(* IEC 61131-3 sources: Word/plc-course/11-program-organization/labs/solutions, 3 files *)

(* ---- 11-1-motor-fb.st ---- *)
(* Lab 11-1: A reusable motor function block, used three times.
   Module 11 (Program organisation). REFERENCE SOLUTION - try the lab yourself first.

   A chemical dosing room has two dosing pumps and an extract fan. One
   function block type, FB_Motor, is written and tested once, then used for
   all three motors. Each instance (Pump1, Pump2, Fan1) has its own memory:
   its own seal-in, its own feedback timer and its own fault latch. *)

FUNCTION_BLOCK FB_Motor
  (* ------------------------------------------------------------------
     FB_Motor - direct-on-line motor with run feedback supervision.

     Behaviour
       - Start (TRUE) switches RunCmd on; RunCmd then holds itself on.
       - Stop, loss of InterlockOK, or a Fault switch RunCmd off. Stop wins
         over Start. The motor never restarts on its own: after a stop, an
         interlock trip or a reset it needs a new Start.
       - RunFb must agree with RunCmd. If they disagree for longer than
         FbTimeout (failed to start, lost feedback while running, or running
         without a command) Fault latches and RunCmd switches off.
       - Reset clears Fault. It does not restart the motor. If the cause is
         still there, the fault comes straight back.
       - Running = commanded AND feedback present ("proven running").
       - RunSeconds counts seconds of proven running (maintenance hours).
         It uses a 1 s timer that restarts every second, so it runs about
         one scan per second slow (1 % at a 10 ms scan). Good enough for
         maintenance hours, not for billing.

     The FB contains no I/O addresses. The calling program maps its inputs
     and outputs to real signals, so the same FB serves any motor.

     Version history
       1.0  first release (Lab 11-1)
     ------------------------------------------------------------------ *)
  VAR_INPUT
    Start       : BOOL;          (* start request, TRUE = start (pulse or held) *)
    Stop        : BOOL;          (* stop request, TRUE = stop; wins over Start *)
    InterlockOK : BOOL;          (* TRUE = allowed to run. No default TRUE on purpose:
                                    a forgotten connection must stop the motor,
                                    not bypass the interlock *)
    RunFb       : BOOL;          (* run feedback: contactor auxiliary contact,
                                    flow switch or airflow switch *)
    Reset       : BOOL;          (* fault reset *)
    FbTimeout   : TIME := T#2s;  (* how long RunFb may disagree with RunCmd *)
  END_VAR
  VAR_OUTPUT
    RunCmd      : BOOL;          (* command to the contactor coil *)
    Running     : BOOL;          (* proven running: RunCmd AND RunFb *)
    Fault       : BOOL;          (* latched feedback fault; needs Reset *)
    RunSeconds  : DINT;          (* extension: seconds of proven running *)
  END_VAR
  VAR
    FbCheck     : TON;           (* feedback discrepancy timer (a multi-instance) *)
    SecondTick  : TON;           (* 1 s time base for RunSeconds *)
  END_VAR

  (* 1. Reset. Checked first, so the discrepancy check further down can set
        the fault again in the same scan if its cause is still present. *)
  IF Reset THEN
    Fault := FALSE;
  END_IF;

  (* 2. Run command: seal-in with stop priority. Stop, interlock and fault
        are tested first, so none of them can be overridden by Start. *)
  IF Stop OR NOT InterlockOK OR Fault THEN
    RunCmd := FALSE;
  ELSIF Start THEN
    RunCmd := TRUE;
  END_IF;

  (* 3. Feedback supervision. XOR is TRUE whenever command and feedback
        disagree: failed to start, feedback lost while running, or running
        without a command (welded contactor, motor run in "hand"). The timer
        restarts every time they agree again. *)
  FbCheck(IN := RunCmd XOR RunFb, PT := FbTimeout);
  IF FbCheck.Q THEN
    Fault := TRUE;
    RunCmd := FALSE;
  END_IF;

  (* 4. Status *)
  Running := RunCmd AND RunFb;

  (* 5. Run-time accumulation (extension). The timer is restarted in the
        same scan that it finishes, so only one scan per second is lost. *)
  SecondTick(IN := Running, PT := T#1s);
  IF SecondTick.Q THEN
    RunSeconds := RunSeconds + 1;
    SecondTick(IN := FALSE);
  END_IF;
END_FUNCTION_BLOCK

PROGRAM DosingRoom
  VAR (* inputs *)
    Pump1StartPB   AT %IX0.0 : BOOL;  (* Pump 1 start push-button, NO *)
    Pump1StopPB_NC AT %IX0.1 : BOOL;  (* Pump 1 stop push-button, NC: TRUE while not pressed *)
    Pump1RunFb     AT %IX0.2 : BOOL;  (* Pump 1 contactor auxiliary contact: TRUE = contactor in *)
    Pump2StartPB   AT %IX0.3 : BOOL;  (* Pump 2 start push-button, NO *)
    Pump2StopPB_NC AT %IX0.4 : BOOL;  (* Pump 2 stop push-button, NC *)
    Pump2RunFb     AT %IX0.5 : BOOL;  (* Pump 2 contactor auxiliary contact *)
    Fan1StartPB    AT %IX0.6 : BOOL;  (* Extract fan start push-button, NO *)
    Fan1StopPB_NC  AT %IX0.7 : BOOL;  (* Extract fan stop push-button, NC *)
    Fan1AirflowSw  AT %IX1.0 : BOOL;  (* Extract duct airflow switch: TRUE = air moving *)
    TankLowLow_NC  AT %IX1.1 : BOOL;  (* Day-tank low-low level switch, fail-safe:
                                         TRUE = level healthy, FALSE = low-low or wire break *)
    ResetPB        AT %IX1.2 : BOOL;  (* Fault reset push-button, NO *)
  END_VAR
  VAR (* outputs *)
    Pump1Contactor AT %QX0.0 : BOOL;  (* Pump 1 contactor coil *)
    Pump2Contactor AT %QX0.1 : BOOL;  (* Pump 2 contactor coil *)
    Fan1Contactor  AT %QX0.2 : BOOL;  (* Extract fan contactor coil *)
    FaultLamp      AT %QX0.3 : BOOL;  (* Common "motor fault" lamp *)
  END_VAR
  VAR (* one instance of FB_Motor per motor *)
    Pump1 : FB_Motor;
    Pump2 : FB_Motor;
    Fan1  : FB_Motor;
  END_VAR

  (* The fan is called first because the pumps use its Running status.
     Calling it after the pumps would also work, one scan later. *)
  Fan1(Start       := Fan1StartPB,
       Stop        := NOT Fan1StopPB_NC,   (* polarity is handled here, not in the FB *)
       InterlockOK := TRUE,                (* the fan has no process interlock *)
       RunFb       := Fan1AirflowSw,
       Reset       := ResetPB,
       FbTimeout   := T#5s);               (* an airflow switch needs a few seconds to prove *)
  Fan1Contactor := Fan1.RunCmd;

  (* Dosing pumps may run only while the extract fan is PROVEN running and
     the day tank is above low-low. Fan1.Running, not Fan1.RunCmd: a fan
     that has been told to run but moves no air does not ventilate the room. *)
  Pump1(Start       := Pump1StartPB,
        Stop        := NOT Pump1StopPB_NC,
        InterlockOK := Fan1.Running AND TankLowLow_NC,
        RunFb       := Pump1RunFb,
        Reset       := ResetPB);           (* FbTimeout left at its 2 s default *)
  Pump1Contactor := Pump1.RunCmd;

  Pump2(Start       := Pump2StartPB,
        Stop        := NOT Pump2StopPB_NC,
        InterlockOK := Fan1.Running AND TankLowLow_NC,
        RunFb       := Pump2RunFb,
        Reset       := ResetPB);
  Pump2Contactor := Pump2.RunCmd;

  FaultLamp := Pump1.Fault OR Pump2.Fault OR Fan1.Fault;
END_PROGRAM

CONFIGURATION Config0
  RESOURCE Res0 ON PLC
    TASK MainTask(INTERVAL := T#10ms, PRIORITY := 0);
    PROGRAM Inst0 WITH MainTask : DosingRoom;
  END_RESOURCE
END_CONFIGURATION

(* ---- 11-2-valve-fb.st ---- *)
(* Lab 11-2: A reusable on/off valve function block with limit switches.
   Module 11 (Program organisation). REFERENCE SOLUTION - try the lab yourself first.

   Two spring-return pneumatic valves on a reactor use the same FB_Valve:
     XV101  reactor feed valve      fail CLOSED (loss of air/power stops the feed)
     XV102  jacket cooling valve    fail OPEN   (loss of air/power keeps cooling on)
   The FB is told which way its valve fails and works out the solenoid state
   for itself. Training exercise only: a real reactor trip belongs in a
   safety instrumented system, not in basic control logic (Module 20). *)

FUNCTION_BLOCK FB_Valve
  (* ------------------------------------------------------------------
     FB_Valve - single-solenoid, spring-return on/off valve with open and
     closed limit switches (ZSO / ZSC).

     Behaviour
       - OpenCmd TRUE = open the valve, FALSE = close it (a level command,
         as a sequence or HMI would give it).
       - FailOpen says where the spring takes the valve when the solenoid is
         de-energised. The solenoid is energised to move the valve AWAY from
         that fail position:  Solenoid = OpenCmd XOR FailOpen.
       - IsOpen / IsClosed are only TRUE when exactly one limit switch is made.
       - TravelFault latches if the valve is not in the commanded end position
         for longer than TravelTime. The timer restarts whenever the command
         changes, so a reversal mid-stroke gets a full TravelTime. It also
         catches a valve that drifts out of position with no command change
         (for example loss of instrument air).
       - LimitFault latches if both limit switches are made together for
         500 ms (a switch, adjustment or wiring fault; the filter ignores a
         momentary overlap).
       - On any fault the solenoid is de-energised, so the valve goes to its
         fail position, and stays there until Reset.
       - Reset clears both faults. After a reset the valve follows OpenCmd
         again and gets a fresh TravelTime. If a fault's cause is still
         present the fault comes back.

     Version history
       1.0  first release (Lab 11-2)
     ------------------------------------------------------------------ *)
  VAR_INPUT
    OpenCmd    : BOOL;            (* TRUE = open, FALSE = close *)
    OpenLS     : BOOL;            (* open limit switch (ZSO), TRUE = fully open *)
    ClosedLS   : BOOL;            (* closed limit switch (ZSC), TRUE = fully closed *)
    Reset      : BOOL;            (* fault reset *)
    FailOpen   : BOOL;            (* configuration: TRUE = spring opens the valve *)
    TravelTime : TIME := T#10s;   (* longest acceptable stroke *)
  END_VAR
  VAR_OUTPUT
    Solenoid    : BOOL;           (* solenoid output *)
    IsOpen      : BOOL;           (* confirmed open *)
    IsClosed    : BOOL;           (* confirmed closed *)
    TravelFault : BOOL;           (* latched: did not reach / stay in position *)
    LimitFault  : BOOL;           (* latched: both limit switches made *)
    Fault       : BOOL;           (* TravelFault OR LimitFault *)
  END_VAR
  VAR
    TravelTmr  : TON;
    LimitTmr   : TON;
    InPosition : BOOL;            (* at the end position the command asks for *)
    LastCmd    : BOOL;            (* OpenCmd on the previous call *)
  END_VAR

  (* 1. Decode the limit switches. Exactly one must be made. *)
  IsOpen := OpenLS AND NOT ClosedLS;
  IsClosed := ClosedLS AND NOT OpenLS;

  (* 2. Reset first, so a fault whose cause is still present re-latches below. *)
  IF Reset THEN
    TravelFault := FALSE;
    LimitFault := FALSE;
  END_IF;

  (* 3. Limit switch discrepancy: both made is physically impossible. *)
  LimitTmr(IN := OpenLS AND ClosedLS, PT := T#500ms);
  IF LimitTmr.Q THEN
    LimitFault := TRUE;
  END_IF;

  (* 4. Travel supervision. The timer runs while the valve is not where it
        was told to be. It is held off for one call when the command changes
        (so it restarts) and while a fault is latched (so that a reset gives
        the valve a fresh TravelTime instead of an instant re-trip). *)
  IF OpenCmd THEN
    InPosition := IsOpen;
  ELSE
    InPosition := IsClosed;
  END_IF;
  TravelTmr(IN := NOT InPosition AND (OpenCmd = LastCmd)
                  AND NOT TravelFault AND NOT LimitFault,
            PT := TravelTime);
  IF TravelTmr.Q THEN
    TravelFault := TRUE;
  END_IF;
  LastCmd := OpenCmd;

  (* 5. Outputs. On a fault the solenoid drops out: the spring takes the
        valve to its fail (safe) position, whichever way that is. *)
  Fault := TravelFault OR LimitFault;
  IF Fault THEN
    Solenoid := FALSE;
  ELSE
    Solenoid := OpenCmd XOR FailOpen;
  END_IF;
END_FUNCTION_BLOCK

PROGRAM ReactorValves
  VAR (* inputs *)
    XV101_OpenSw AT %IX0.0 : BOOL;  (* XV-101 panel selector: TRUE = OPEN, FALSE = CLOSE *)
    XV101_ZSO    AT %IX0.1 : BOOL;  (* XV-101 open limit switch *)
    XV101_ZSC    AT %IX0.2 : BOOL;  (* XV-101 closed limit switch *)
    XV102_OpenSw AT %IX0.3 : BOOL;  (* XV-102 panel selector: TRUE = OPEN, FALSE = CLOSE *)
    XV102_ZSO    AT %IX0.4 : BOOL;  (* XV-102 open limit switch *)
    XV102_ZSC    AT %IX0.5 : BOOL;  (* XV-102 closed limit switch *)
    ResetPB      AT %IX0.6 : BOOL;  (* Fault reset push-button, NO *)
  END_VAR
  VAR (* outputs *)
    XV101_SOL    AT %QX0.0 : BOOL;  (* XV-101 solenoid: energise to OPEN (fail closed) *)
    XV102_SOL    AT %QX0.1 : BOOL;  (* XV-102 solenoid: energise to CLOSE (fail open) *)
    FaultLamp    AT %QX0.2 : BOOL;  (* Common "valve fault" lamp *)
  END_VAR
  VAR (* device instances *)
    XV101 : FB_Valve;               (* reactor feed valve *)
    XV102 : FB_Valve;               (* jacket cooling-water valve *)
  END_VAR

  XV101(OpenCmd    := XV101_OpenSw,
        OpenLS     := XV101_ZSO,
        ClosedLS   := XV101_ZSC,
        Reset      := ResetPB,
        FailOpen   := FALSE,        (* spring closes it: stop feeding on loss of air *)
        TravelTime := T#5s);
  XV101_SOL := XV101.Solenoid;

  XV102(OpenCmd    := XV102_OpenSw,
        OpenLS     := XV102_ZSO,
        ClosedLS   := XV102_ZSC,
        Reset      := ResetPB,
        FailOpen   := TRUE,         (* spring opens it: keep cooling on loss of air *)
        TravelTime := T#8s);        (* larger valve, slower actuator *)
  XV102_SOL := XV102.Solenoid;

  FaultLamp := XV101.Fault OR XV102.Fault;
END_PROGRAM

CONFIGURATION Config0
  RESOURCE Res0 ON PLC
    TASK MainTask(INTERVAL := T#10ms, PRIORITY := 0);
    PROGRAM Inst0 WITH MainTask : ReactorValves;
  END_RESOURCE
END_CONFIGURATION

(* ---- 11-3-function-library.st ---- *)
(* Lab 11-3: A small function library and a statistics FB using VAR_IN_OUT.
   Module 11 (Program organisation). REFERENCE SOLUTION - try the lab yourself first.

   A filling line has two filling heads, each with its own check-weigher.
   One instance of FB_SampleStats per head judges each weight against the
   limits and adds it to ONE shared statistics record, LineStats, which the
   instances reach through VAR_IN_OUT. Two FUNCTIONs form a small reusable
   library: F_InRange (limit check) and F_Deadband (report-by-exception). *)

TYPE
  ST_Stats :
  STRUCT
    Count    : DINT;    (* samples since the last clear *)
    InSpec   : DINT;    (* samples inside the limits *)
    OutSpec  : DINT;    (* samples outside the limits *)
    MinValue : REAL;    (* smallest sample since the last clear *)
    MaxValue : REAL;    (* largest sample since the last clear *)
    Sum      : LREAL;   (* running total. LREAL: a REAL has only about 7 significant
                           digits. Once a REAL total passes about 8.4 million (some
                           17,000 samples of 500 g) it can only change in whole grams,
                           so every new weight would be rounded to a whole gram *)
    Mean     : REAL;    (* Sum / Count *)
  END_STRUCT;
END_TYPE

FUNCTION F_InRange : BOOL
  (* TRUE when Low <= Value <= High (both limits included).
     If Low > High the range is empty and the result is always FALSE, so a
     limit entry mistake shows up as "everything out of range" rather than
     being silently repaired. No memory: same inputs, same answer. *)
  VAR_INPUT
    Value : REAL;
    Low   : REAL;
    High  : REAL;
  END_VAR
  F_InRange := (Value >= Low) AND (Value <= High);
END_FUNCTION

FUNCTION F_Deadband : REAL
  (* Report-by-exception: returns NewValue when it differs from OldValue by
     Band or more, otherwise returns OldValue unchanged.
     A function has no memory, so the CALLER keeps the last reported value
     and passes it back in as OldValue:
         Reported := F_Deadband(Live, Reported, 0.5);
     Band <= 0.0 passes every change straight through. *)
  VAR_INPUT
    NewValue : REAL;   (* live value *)
    OldValue : REAL;   (* value reported last time *)
    Band     : REAL;   (* smallest change worth reporting *)
  END_VAR
  IF ABS(NewValue - OldValue) >= Band THEN
    F_Deadband := NewValue;
  ELSE
    F_Deadband := OldValue;
  END_IF;
END_FUNCTION

FUNCTION_BLOCK FB_SampleStats
  (* Adds one sample to a statistics record on each rising edge of Sample.
     The record itself is NOT inside the FB: it is passed in by reference
     (VAR_IN_OUT), so several instances can update one shared record and
     the caller decides where it lives (retentive memory, HMI area, ...).
     What IS inside the instance: its own edge detector, its own Reject
     output and its own sample counter. *)
  VAR_INPUT
    Sample    : BOOL;   (* rising edge = Value holds a new sample *)
    Value     : REAL;
    LowLimit  : REAL;
    HighLimit : REAL;
  END_VAR
  VAR_IN_OUT
    Stats     : ST_Stats;
  END_VAR
  VAR_OUTPUT
    Reject    : BOOL;   (* TRUE when this instance's latest sample was out of limits *)
    Samples   : DINT;   (* samples taken by THIS instance since power-up *)
  END_VAR
  VAR
    SampleEdge : R_TRIG;
  END_VAR

  SampleEdge(CLK := Sample);
  IF SampleEdge.Q THEN
    Samples := Samples + 1;

    (* The first sample after a clear seeds MIN and MAX. Starting them at 0.0
       would leave MinValue stuck at 0.0 for ever. *)
    IF Stats.Count = 0 THEN
      Stats.MinValue := Value;
      Stats.MaxValue := Value;
    ELSE
      Stats.MinValue := MIN(Stats.MinValue, Value);
      Stats.MaxValue := MAX(Stats.MaxValue, Value);
    END_IF;

    Stats.Count := Stats.Count + 1;
    Stats.Sum := Stats.Sum + REAL_TO_LREAL(Value);
    Stats.Mean := LREAL_TO_REAL(Stats.Sum / DINT_TO_LREAL(Stats.Count));  (* Count >= 1 here *)

    IF F_InRange(Value, LowLimit, HighLimit) THEN
      Stats.InSpec := Stats.InSpec + 1;
      Reject := FALSE;
    ELSE
      Stats.OutSpec := Stats.OutSpec + 1;
      Reject := TRUE;
    END_IF;
  END_IF;
END_FUNCTION_BLOCK

PROGRAM CheckWeigher
  VAR (* inputs *)
    Head1Ready  AT %IX0.0 : BOOL;  (* check-weigher 1: TRUE when Head1Weight holds a new weight *)
    Head2Ready  AT %IX0.1 : BOOL;  (* check-weigher 2: TRUE when Head2Weight holds a new weight *)
    ClearPB     AT %IX0.2 : BOOL;  (* clear the line statistics (start of shift) *)
  END_VAR
  VAR (* outputs *)
    Head1Reject AT %QX0.0 : BOOL;  (* reject gate after head 1 *)
    Head2Reject AT %QX0.1 : BOOL;  (* reject gate after head 2 *)
  END_VAR
  VAR (* weights from the check-weighers and settings from the HMI *)
    Head1Weight  : REAL;             (* g, written by check-weigher 1 over the network *)
    Head2Weight  : REAL;             (* g, written by check-weigher 2 *)
    LowLimit     : REAL := 495.0;    (* g, lowest acceptable net weight *)
    HighLimit    : REAL := 505.0;    (* g, highest acceptable net weight *)
    MeanDeadband : REAL := 0.5;      (* g, smallest change of mean worth sending to SCADA *)
  END_VAR
  VAR (* data *)
    LineStats    : ST_Stats;         (* shared by both heads, read by the HMI *)
    ReportedMean : REAL;             (* mean weight as last sent to SCADA *)
    Head1        : FB_SampleStats;
    Head2        : FB_SampleStats;
  END_VAR
  VAR CONSTANT
    (* A record with every field at zero, for clearing LineStats in one
       assignment. Every member of ST_Stats starts at 0 or 0.0 anyway, so no
       initialiser is needed. Writing one out, (Count := 0, ..., Mean := 0.0),
       is standard IEC 61131-3, but OpenPLC's compiler does not accept this
       initialiser (see Appendix E). *)
    CLEARED_STATS : ST_Stats;
  END_VAR

  (* Both instances update the SAME record. VAR_IN_OUT must be connected
     to a variable on every call; a constant or an expression is refused. *)
  Head1(Sample := Head1Ready, Value := Head1Weight,
        LowLimit := LowLimit, HighLimit := HighLimit,
        Stats := LineStats);
  Head2(Sample := Head2Ready, Value := Head2Weight,
        LowLimit := LowLimit, HighLimit := HighLimit,
        Stats := LineStats);

  (* Clear AFTER the calls: the record then reads all zeros for as long as
     ClearPB is held, even if a weight arrives in that scan. Such a weight
     still operates its reject gate; it is just not added to the new shift. *)
  IF ClearPB THEN
    LineStats := CLEARED_STATS;
  END_IF;

  Head1Reject := Head1.Reject;
  Head2Reject := Head2.Reject;

  (* ReportedMean is the memory that F_Deadband itself cannot have. *)
  ReportedMean := F_Deadband(LineStats.Mean, ReportedMean, MeanDeadband);
END_PROGRAM

CONFIGURATION Config0
  RESOURCE Res0 ON PLC
    TASK MainTask(INTERVAL := T#10ms, PRIORITY := 0);
    PROGRAM Inst0 WITH MainTask : CheckWeigher;
  END_RESOURCE
END_CONFIGURATION
